IF ResetMethodCall THEN
    MethodCall_RotationMove := FALSE;
    jobRunning := FALSE;
    jobFinished := TRUE;
    state := 100;
END_IF;
                

{attribute 'TcRpcEnable' := '1'}
METHOD Abort : HRESULT
VAR_INPUT
    hdl : UDINT;
END_VAR
                        callCounterAbort := callCounterAbort + 1;

MethodCall_RotationMove := FALSE;
DO_MovingRotationVSG_01 := FALSE;

jobRunning := FALSE;
jobFinished := TRUE;
state := 999;

Abort := 0;
                      
END_METHOD

{attribute 'TcRpcEnable' := '1'}
METHOD CheckState : HRESULT
VAR_INPUT
    hdl : UDINT;
END_VAR

VAR_OUTPUT
    bBusy : BOOL;
    State : UDINT;
    IsDone : BOOL;
END_VAR
                        callCounterCheckState := callCounterCheckState + 1;

bBusy := jobRunning;
State := state;
IsDone := jobFinished;

CheckState := 0;
                      
END_METHOD

{attribute 'TcRpcEnable' := '1'}
METHOD Start : HRESULT
VAR_INPUT
    MethodCall : BOOL;
    MovementDirection : BOOL;
    EncoderPositionRotation_01 : UDINT;
    EncoderPositionRotation_02 : UDINT;
    TouchSensorRelief : BOOL;
END_VAR

VAR_OUTPUT
    hdl : UDINT;
END_VAR
                        callCounterStart := callCounterStart + 1;

IF NOT jobRunning THEN

    MethodCall_RotationMove := MethodCall;
    DirectionRotation := MovementDirection;

    EncoderTargetPosition01 := EncoderPositionRotation_01;
    EncoderTargetPosition02 := EncoderPositionRotation_02;

    TSR := TouchSensorRelief;

    jobRunning := TRUE;
    jobFinished := FALSE;
    state := 1;

    hdl := 1;
    Start := 0;

ELSE

    hdl := 0;
    Start := 16#800700AA;

END_IF;
                      
END_METHOD
END_FUNCTION_BLOCK

{attribute 'OPC.UA.DA.JobMethod' := 'JobMethode_VerticalMove'}
FUNCTION_BLOCK VSG_AS_VerticalMoveEncoder
VAR
    MethodCall_VerticalMove : BOOL := FALSE;
    ResetMethodCall : BOOL := FALSE;

    DirectionVertical : BOOL := TRUE;

    EncoderTargetPosition01 : UDINT;
    EncoderTargetPosition02 : UDINT;

    TSR : BOOL := FALSE;

    callCounterStart : ULINT;
    callCounterCheckState : ULINT;
    callCounterAbort : ULINT;

    jobRunning : BOOL := FALSE;
    jobFinished : BOOL := FALSE;
    state : UDINT := 0;

    VSG_VerticalMoveWithEncoder : AxisControl_Encoder;
END_VAR

VAR_INPUT
    ESS : BOOL;
    TouchSensor01 : BOOL;
    EncoderStartPosition01 : UDINT;
    EncoderStartPosition02 : UDINT;
    TOF_Time_TSR : TIME;
    AutomaticMode : BOOL;
END_VAR

VAR_OUTPUT
    DO_MovingVerticalVSG_01 : BOOL;
END_VAR

                  VSG_VerticalMoveWithEncoder(
    MethodCall := MethodCall_VerticalMove,
    EmergencyStopSignal := NOT ESS,
    Direction := DirectionVertical,
    InitStateDrive_Input := FALSE,
    DI01 := TouchSensor01,
    DI02_EncoderStart01 := EncoderStartPosition01,
    DI03_EncoderTarget01 := EncoderTargetPosition01,
    DI04_EncoderStart02 := EncoderStartPosition02,
    DI05_EncoderTarget02 := EncoderTargetPosition02,
    TouchSensorRelief := TSR,
    TOF_Time_MotorControl := T#0MS,
    TOF_Time_TouchSensorRelief := TOF_Time_TSR,
    OperatingMode := AutomaticMode
);

DO_MovingVerticalVSG_01 := VSG_VerticalMoveWithEncoder.DigitalOutputControl_01;
ResetMethodCall := VSG_VerticalMoveWithEncoder.ResetMethodCall;

IF ResetMethodCall THEN
    MethodCall_VerticalMove := FALSE;
    jobRunning := FALSE;
    jobFinished := TRUE;
    state := 100;
END_IF;
                

{attribute 'TcRpcEnable' := '1'}
METHOD Abort : HRESULT
VAR_INPUT
    hdl : UDINT;
END_VAR
                        callCounterAbort := callCounterAbort + 1;

MethodCall_VerticalMove := FALSE;
DO_MovingVerticalVSG_01 := FALSE;

jobRunning := FALSE;
jobFinished := TRUE;
state := 999;

Abort := 0;
                      
END_METHOD

{attribute 'TcRpcEnable' := '1'}
METHOD CheckState : HRESULT
VAR_INPUT
    hdl : UDINT;
END_VAR

VAR_OUTPUT
    bBusy : BOOL;
    State : UDINT;
    IsDone : BOOL;
END_VAR
                        callCounterCheckState := callCounterCheckState + 1;

bBusy := jobRunning;
State := state;
IsDone := jobFinished;

CheckState := 0;
                      
END_METHOD

{attribute 'TcRpcEnable' := '1'}
METHOD Start : HRESULT
VAR_INPUT
    MethodCall : BOOL;
    MovementDirection : BOOL;
    EncoderPositionVertical_01 : UDINT;
    EncoderPositionVertical_02 : UDINT;
    TouchSensorRelief : BOOL;
END_VAR

VAR_OUTPUT
    hdl : UDINT;
END_VAR
                        callCounterStart := callCounterStart + 1;

IF NOT jobRunning THEN

    MethodCall_VerticalMove := MethodCall;
    DirectionVertical := MovementDirection;

    EncoderTargetPosition01 := EncoderPositionVertical_01;
    EncoderTargetPosition02 := EncoderPositionVertical_02;

    TSR := TouchSensorRelief;

    jobRunning := TRUE;
    jobFinished := FALSE;
    state := 1;

    hdl := 1;
    Start := 0;

ELSE

    hdl := 0;
    Start := 16#800700AA;

END_IF;
                      
END_METHOD
END_FUNCTION_BLOCK

CONFIGURATION Application
  RESOURCE SPS_Demonstrator ON PLC
(* global variable list GVL *)
{attribute 'qualified_only'}
VAR_GLOBAL
	// xDI%139.2_S1_2
	diNotAus_Kanal_A AT %I*: BOOL;
	// xDI%139.3_S1_2
	diNotAus_Kanal_B AT %I*: BOOL;
END_VAR
(* global variable list GVL_HRL *)
{attribute 'qualified_only'}
VAR_GLOBAL
	// udiDI%41.0_A2_5
	{attribute 'OPC.UA.DA' := '1'} // für OPC UA freigeben
	HRL_Enc_horizontal_I1 AT %I*: UDINT;
	{attribute 'OPC.UA.DA' := '1'} // für OPC UA freigeben
	// udiDI%47.0_A2_5
	HRL_Enc_horizontal_I2 AT %I*: UDINT;
	{attribute 'OPC.UA.DA' := '1'} // für OPC UA freigeben
	// udiDI%53.0_A2_5
	HRL_Enc_vertikal_I1 AT %I*: UDINT;
	{attribute 'OPC.UA.DA' := '1'} // für OPC UA freigeben
	// udiDI%59.0_A2_5
	HRL_Enc_vertikal_I2 AT %I*: UDINT;
	{attribute 'OPC.UA.DA' := '1'} // für OPC UA freigeben
	// xDI%136.0_A2_2
	HRL_Ref_Taster_horizontal AT %I*: BOOL;
	{attribute 'OPC.UA.DA' := '1'} // für OPC UA freigeben
	// xDI%136.1_A2_1
	{attribute 'OPC.UA.DA' := '1'} // für OPC UA freigeben
	HRL_LS_innen AT %I*: BOOL;
	// xDI%136.2_A2_1
	{attribute 'OPC.UA.DA' := '1'} // für OPC UA freigeben
	HRL_LS_aussen AT %I*: BOOL;
	// xDI%136.3_A2_2
	{attribute 'OPC.UA.DA' := '1'} // für OPC UA freigeben
	HRL_Ref_Taster_vertikal AT %I*: BOOL;
	// xDI%136.4_A2_3
	{attribute 'OPC.UA.DA' := '1'} // für OPC UA freigeben
	HRL_Spursensor_1_unten AT %I*: BOOL;
	// xDI%136.5_A2_3
	{attribute 'OPC.UA.DA' := '1'} // für OPC UA freigeben
	HRL_Spursensor_2_oben AT %I*: BOOL;
	// xDI%136.6_A2_2
	{attribute 'OPC.UA.DA' := '1'} // für OPC UA freigeben
	HRL_Ref_Taster_Ausleger_vorne AT %I*: BOOL;
	// xDI%136.7_A2_2
	{attribute 'OPC.UA.DA' := '1'} // für OPC UA freigeben
	HRL_Ref_Taster_Ausleger_hinten AT %I*: BOOL;
	// xDO%111.0_A2_2	
	{attribute 'OPC.UA.DA' := '1'} // für OPC UA freigeben
	HRL_MOT_Foerderband_vorwaerts AT %Q*: BOOL;
	// xDO%111.1_A2_2
	{attribute 'OPC.UA.DA' := '1'} // für OPC UA freigeben
	HRL_MOT_Foerderband_rueckwaerts AT %Q*: BOOL;
	// xDO%111.2_A2_4
	{attribute 'OPC.UA.DA' := '1'} // für OPC UA freigeben
	HRL_MOT_horizontal_zum_Regal AT %Q*: BOOL;
	// xDO%111.3_A2_4
	{attribute 'OPC.UA.DA' := '1'} // für OPC UA freigeben
	HRL_MOT_horizontal_zum_Foerderband AT %Q*: BOOL;
	// xDO%111.4_A2_4
	{attribute 'OPC.UA.DA' := '1'} // für OPC UA freigeben
	HRL_MOT_vertikal_runter AT %Q*: BOOL;
	// xDO%111.5_A2_4
	{attribute 'OPC.UA.DA' := '1'} // für OPC UA freigeben
	HRL_MOT_vertikal_hoch AT %Q*: BOOL;
	// xDO%111.6_A2_4
	{attribute 'OPC.UA.DA' := '1'} // für OPC UA freigeben
	HRL_MOT_Ausleger_vorwaerts AT %Q*: BOOL;
	// xDO%111.7_A2_4
	{attribute 'OPC.UA.DA' := '1'} // für OPC UA freigeben
	HRL_MOT_Ausleger_rueckwaerts AT %Q*: BOOL;
	{attribute 'OPC.UA.DA' := '1'} // für OPC UA freigeben
	HRL_K1_1_Zaehler_Zuruecksetzen AT %Q*: BOOL;
	{attribute 'OPC.UA.DA' := '1'} // für OPC UA freigeben
	HRL_K1_2_Zaehler_Zuruecksetzen AT %Q*: BOOL;
END_VAR
(* global variable list GVL_HRL_Sim *)
{attribute 'qualified_only'}
VAR_GLOBAL
	// Spiegel von GVL_HRL (Eingänge)
    HRL_Enc_horizontal_I1 : UDINT;
	// udiDI%47.0_A2_5
	HRL_Enc_horizontal_I2 : UDINT;
	// udiDI%53.0_A2_5
	HRL_Enc_vertikal_I1 : UDINT;
	// udiDI%59.0_A2_5
	HRL_Enc_vertikal_I2 : UDINT;
	// xDI%136.0_A2_2
	HRL_Ref_Taster_horizontal : BOOL;
	// xDI%136.1_A2_1
	HRL_LS_innen : BOOL;
	// xDI%136.2_A2_1
	HRL_LS_aussen : BOOL;
	// xDI%136.3_A2_2
	HRL_Ref_Taster_vertikal : BOOL;
	// xDI%136.4_A2_3
	HRL_Spursensor_1_unten : BOOL;
	// xDI%136.5_A2_3
	HRL_Spursensor_2_oben : BOOL;
	// xDI%136.6_A2_2
	HRL_Ref_Taster_Ausleger_vorne : BOOL;
	// xDI%136.7_A2_2
	HRL_Ref_Taster_Ausleger_hinten : BOOL;
	// xDO%111.0_A2_2	
	HRL_MOT_Foerderband_vorwaerts : BOOL;
	// xDO%111.1_A2_2
	HRL_MOT_Foerderband_rueckwaerts : BOOL;
	// xDO%111.2_A2_4
	HRL_MOT_horizontal_zum_Regal : BOOL;
	// xDO%111.3_A2_4
	HRL_MOT_horizontal_zum_Foerderband : BOOL;
	// xDO%111.4_A2_4
	HRL_MOT_vertikal_runter : BOOL;
	// xDO%111.5_A2_4
	HRL_MOT_vertikal_hoch : BOOL;
	// xDO%111.6_A2_4
	HRL_MOT_Ausleger_vorwaerts : BOOL;
	// xDO%111.7_A2_4
	HRL_MOT_Ausleger_rueckwaerts : BOOL;
	HRL_K1_1_Zaehler_Zuruecksetzen : BOOL;
	HRL_K1_2_Zaehler_Zuruecksetzen : BOOL;
END_VAR
(* global variable list GVL_MBS *)
{attribute 'qualified_only'}
VAR_GLOBAL
	// xDI%137.0_A3_2
	MBS_Ref_Taster_DK_Pos_Sauger AT %I*: BOOL;
	// xDI%137.1_A3_2
	MBS_Ref_Taster_DK_Pos_Foerderband AT %I*: BOOL;
	// xDI%137.2_A3_1
	MBS_LS_Ende_Foerderband AT %I*: BOOL;
	// xDI%137.3_A3_2
	MBS_Ref_Taster_DK_Pos_Saege AT %I*: BOOL;
	// xDI%137.4_A3_2
	MBS_Ref_Taster_Sauger_Pos_DK AT %I*: BOOL;
	// xDI%137.5_A3_2
	MBS_Ref_Taster_Ofenschieber_innen AT %I*: BOOL;
	// xDI%137.6_A3_2
	MBS_Ref_Taster_Ofenschieber_aussen AT %I*: BOOL;
	// xDI%137.7_A3_2
	MBS_Ref_Taster_Sauger_Pos_Ofen AT %I*: BOOL;
	// xDI%138.0_A3_1
	MBS_LS_Ofen AT %I*: BOOL;
	// xDO%112.0_A3_4
	MBS_MOT_DK_CW AT %Q*: BOOL;
	// xDO%112.1_A3_4
	MBS_MOT_DK_CCW AT %Q*: BOOL;
	// xDO%112.2_A3_2
	MBS_MOT_Foerderband_vorwaerts AT %Q*: BOOL;
	// xDO%112.3_A3_6
	MBS_MOT_Saege AT %Q*: BOOL;
	// xDO%112.4_A3_3
	MBS_MOT_Ofenschieber_einfahren AT %Q*: BOOL;
	// xDO%112.5_A3_3
	MBS_MOT_Ofenschieber_ausfahren AT %Q*: BOOL;
	// xDO%112.6_A3_5
	MBS_MOT_Sauger_zum_Ofen AT %Q*: BOOL;
	// xDO%112.7_A3_5
	MBS_MOT_Sauger_zum_DK AT %Q*: BOOL;
	// xDO%113.0_A3_7
	MBS_Leuchte_Ofen AT %Q*: BOOL;
	// xDO%113.1_A3_8
	MBS_Kompressor AT %Q*: BOOL;
	// xDO%113.2_A3_5
	MBS_MV_Vakuum AT %Q*: BOOL;
	// xDO%113.3_A3_5
	MBS_MV_senken AT %Q*: BOOL;
	// xDO%113.4_A3_5
	MBS_MV_Ofentuer AT %Q*: BOOL;
	// xDO%113.5_A3_5
	MBS_MV_Schieber AT %Q*: BOOL;
END_VAR
(* global variable list GVL_Sim *)
{attribute 'qualified_only'}
VAR_GLOBAL
	bSimMode : BOOL ;   // FALSE = reale Hardware, TRUE = Python-Simulation

    // Spiegel von GVL
    diNotAus_Kanal_A : BOOL ;
    diNotAus_Kanal_B : BOOL ;
    
END_VAR
(* global variable list GVL_SST *)
{attribute 'qualified_only'}
VAR_GLOBAL
	// xDO%115.0_A5_5
	SST_MV_weiss AT %Q*: BOOL;
	// xDO%115.1_A5_5
	SST_MV_rot AT %Q*: BOOL;
	// xDO%115.2_A5_5
	SST_MV_blau AT %Q*: BOOL;
	// iAI%130.0_A5_4
	SST_Farbsensor AT %I*: INT;
	// xDI%138.4_A5_1
	SST_Impulstaster AT %I*: BOOL;
	// xDI%138.5_A5_1
	SST_LS_Eingang AT %I*: BOOL;
	// xDI%138.6_A5_1
	SST_LS_nach_Farbsensor AT %I*: BOOL;
	// xDI%138.7_A5_1
	SST_LS_weiss AT %I*: BOOL;
	// xDI%139.0_A5_1
	SST_LS_rot AT %I*: BOOL;
	// xDI%139.1_A5_1
	SST_LS_blau AT %I*: BOOL;
	// xDO%114.6_A5_2
	SST_MOT_Foerderband AT %Q*: BOOL;
	// xDO%114.7_A5_8
	SST_Kompressor AT %Q*: BOOL;
END_VAR
(* global variable list GVL_VSG *)
{attribute 'qualified_only'}
VAR_GLOBAL
	// udiDI%65.0_A4_5
	{attribute 'OPC.UA.DA' := '1'} // für OPC UA freigeben
	VSG_Enc_vertikal_I1 AT %I*: UDINT;
	{attribute 'OPC.UA.DA' := '1'} // für OPC UA freigeben
	// udiDI%71.0_A4_5
	VSG_Enc_vertikal_I2 AT %I*: UDINT;
	{attribute 'OPC.UA.DA' := '1'} // für OPC UA freigeben
	// udiDI%77.0_A4_5
	VSG_Enc_horizontal_I1 AT %I*: UDINT;
	{attribute 'OPC.UA.DA' := '1'} // für OPC UA freigeben
	// udiDI%83.0_A4_5
	VSG_Enc_horizontal_I2 AT %I*: UDINT;
	{attribute 'OPC.UA.DA' := '1'} // für OPC UA freigeben
	// udiDI%89.0_A4_5
	VSG_Enc_drehen_I1 AT %I*: UDINT;
	{attribute 'OPC.UA.DA' := '1'} // für OPC UA freigeben
	// udiDI%95.0_A4_5
	VSG_Enc_drehen_I2 AT %I*: UDINT;
	{attribute 'OPC.UA.DA' := '1'} // für OPC UA freigeben
	// xDI%138.1_A4_2
	VSG_Ref_Schalter_vertikal AT %I*: BOOL;
	{attribute 'OPC.UA.DA' := '1'} // für OPC UA freigeben
	// xDI%138.2_A4_2
	VSG_Ref_Schalter_horizontal AT %I*: BOOL;
	{attribute 'OPC.UA.DA' := '1'} // für OPC UA freigeben
	// xDI%138.3_A4_2
	VSG_Ref_Schalter_drehen AT %I*: BOOL;
	{attribute 'OPC.UA.DA' := '1'} // für OPC UA freigeben
	// xDO%113.6_A4_4
	VSG_MOT_vertikal_hoch AT %Q*: BOOL;
	{attribute 'OPC.UA.DA' := '1'} // für OPC UA freigeben
	// xDO%113.7_A4_4
	VSG_MOT_vertikal_runter AT %Q*: BOOL;
	{attribute 'OPC.UA.DA' := '1'} // für OPC UA freigeben
	// xDO%114.0_A4_4
	VSG_MOT_horizontal_rueckwaerts AT %Q*: BOOL;
	{attribute 'OPC.UA.DA' := '1'} // für OPC UA freigeben
	// xDO%114.1_A4_4
	VSG_MOT_horizontal_vorwaerts AT %Q*: BOOL;
	{attribute 'OPC.UA.DA' := '1'} // für OPC UA freigeben
	// xDO%114.2_A4_4
	VSG_MOT_drehen_CW AT %Q*: BOOL;
	{attribute 'OPC.UA.DA' := '1'} // für OPC UA freigeben
	// xDO%114.3_A4_4
	VSG_MOT_drehen_CCW AT %Q*: BOOL;
	{attribute 'OPC.UA.DA' := '1'} // für OPC UA freigeben
	// xDO%114.4_A4_8
	VSG_Kompressor AT %Q*: BOOL;
	{attribute 'OPC.UA.DA' := '1'} // für OPC UA freigeben
	// xDO%114.5_A4_5
	{attribute 'OPC.UA.DA' := '1'} // für OPC UA freigeben
	VSG_MV_Vakuum AT %Q*: BOOL;
	{attribute 'OPC.UA.DA' := '1'} // für OPC UA freigeben
	VSG_K1_4_Zaehler_Zuruecksetzen AT %Q*: BOOL;
	{attribute 'OPC.UA.DA' := '1'} // für OPC UA freigeben
	VSG_K1_5_Zaehler_Zuruecksetzen AT %Q*: BOOL;
	{attribute 'OPC.UA.DA' := '1'} // für OPC UA freigeben
	VSG_K1_3_Zaehler_Zuruecksetzen AT %Q*: BOOL;
END_VAR
(* global variable list GVL_VSG_Sim *)
{attribute 'qualified_only'}
VAR_GLOBAL
    // Simulierte VSG Eingänge
    VSG_Enc_vertikal_I1 : UDINT;
    VSG_Enc_vertikal_I2 : UDINT;

    VSG_Enc_horizontal_I1 : UDINT;
    VSG_Enc_horizontal_I2 : UDINT;

    VSG_Enc_drehen_I1 : UDINT;
    VSG_Enc_drehen_I2 : UDINT;

    VSG_Ref_Schalter_vertikal : BOOL;
    VSG_Ref_Schalter_horizontal : BOOL;
    VSG_Ref_Schalter_drehen : BOOL;

    // Simulierte VSG Ausgänge
    VSG_MOT_vertikal_hoch : BOOL;
    VSG_MOT_vertikal_runter : BOOL;

    VSG_MOT_horizontal_vorwaerts : BOOL;
    VSG_MOT_horizontal_rueckwaerts : BOOL;

    VSG_MOT_drehen_CW : BOOL;
    VSG_MOT_drehen_CCW : BOOL;

    VSG_Kompressor : BOOL;
    VSG_MV_Vakuum : BOOL;

    VSG_K1_4_Zaehler_Zuruecksetzen : BOOL;
    VSG_K1_5_Zaehler_Zuruecksetzen : BOOL;
    VSG_K1_3_Zaehler_Zuruecksetzen : BOOL;
END_VAR
(* global variable list OPCUA *)
{attribute 'qualified_only'}
VAR_GLOBAL
	{attribute 'OPC.UA.DA' := '1'} // für OPC UA freigeben
	TriggerD1 : BOOL := FALSE;
	{attribute 'OPC.UA.DA' := '1'} // für OPC UA freigeben
	TriggerD2 : BOOL := FALSE;
	{attribute 'OPC.UA.DA' := '1'} // für OPC UA freigeben
	TriggerD3 : BOOL := FALSE;
	{attribute 'OPC.UA.DA' := '1'} // für OPC UA freigeben
    {attribute 'OPC.UA.DA.Access' := '3'} // Read/Write
	Alt_found : BOOL := FALSE;
	{attribute 'OPC.UA.DA' := '1'} // für OPC UA freigeben
    {attribute 'OPC.UA.DA.Access' := '3'} // Read/Write
	Alt_abort : BOOL := FALSE;
	{attribute 'OPC.UA.DA' := '1'} // für OPC UA freigeben
    {attribute 'OPC.UA.DA.Access' := '3'} // Read/Write
	Diag_finished : BOOL := FALSE;
	{attribute 'OPC.UA.DA' := '1'} // für OPC UA freigeben
    {attribute 'OPC.UA.DA.Access' := '3'} // Read/Write
	Cycle_finished : BOOL := FALSE;
	{attribute 'OPC.UA.DA' := '1'}
    LastGEMMAStateBeforeFailure: STRING;
	{attribute 'OPC.UA.DA' := '1'}
    lastExecutedSkill: STRING := '';
	{attribute 'OPC.UA.DA' := '1'}
	{attribute 'OPC.UA.DA.Access' := '3'} // Read/Write
    lastFinishedSkill: STRING := '';
	{attribute 'OPC.UA.DA' := '1'}
    lastExecutedProcess: STRING := '';
END_VAR
    TASK PlcTask(INTERVAL := T#0ms, PRIORITY := 20);
    PROGRAM HRL_SkillSet WITH PlcTask : HRL_SkillSet;
    PROGRAM VSG_SkillSet WITH PlcTask : VSG_SkillSet;
  END_RESOURCE
END_CONFIGURATION
